Fanuc KAREL source: kt00037.KL

-- PROVISIONAL review KL for V770-1; original PC SHA256 f89ed7fdf20bea6f690e5a1cf5bfb521377227db49d307d753e5e1a054da1e01
-- Incomplete behavior may be omitted. Consult companion uncertainty JSON. Do not deploy.
PROGRAM KT00037
%NOLOCKGROUP
VAR
  I1 : INTEGER
  OUT : INTEGER
-- UNRESOLVED_DECL Y2 type=002018
BEGIN
  -- UNRESOLVED_PC offsets 5-16; opcodes 2E,23
  -- UNRESOLVED_PC offsets 21-35; opcodes 2E,22,9D,33,B2
  -- UNRESOLVED_PC offsets 40-62; opcodes 21,22,9D,33,B1,53,23
  -- UNRESOLVED_PC offsets 67-71; opcodes 7F
END KT00037
